TYPE ST_GantrySysPar :
STRUCT
	HorizontalAxis				: ST_NcAxis_SysPar;
	VerticalAxis				: ST_NcAxis_SysPar;	
END_STRUCT
END_TYPE

(* stored: Version 1.1.0.1, ProductVersion 3.1.4020.12
   DUT ST_GantrySysPar: Id {d31372a8-5efe-48c9-911e-b83f9690f168} *)
